FUNCTION_BLOCK ResetStopCounter (* Basic Function Block Type *)
  (* Standard: 61499-2 *)
  (* Version 0.0, 7/16/2026, Schneider Electric, Template *)
  PACKAGE SE.Nereda;
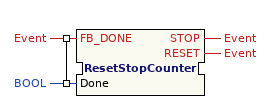
  EVENT_INPUT
    FB_DONE WITH Done; (* Normal Execution Request *)
  END_EVENT
  EVENT_OUTPUT
    STOP;
    RESET;
  END_EVENT
  VAR_INPUT
    Done : BOOL; (* Input event qualifier *)
  END_VAR
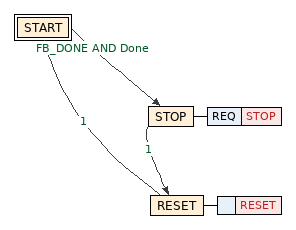
  EC_STATES
    START; (* Initial State *)
    STOP : REQ -> STOP; (* Normal execution *)
    RESET : -> RESET;
  END_STATES
  EC_TRANSITIONS
    START TO STOP := FB_DONE AND Done;
    STOP TO RESET := 1;
    RESET TO START := 1;
  END_TRANSITIONS
  ALGORITHM REQ IN ST: (* Normally executed algorithm *)
;
  END_ALGORITHM
END_FUNCTION_BLOCK
